(* CoDeSys 2.3 export: A_CONV.EXP *)

(* POU A_CONVER, CFC *)
FUNCTION_BLOCK A_CONVER
VAR_INPUT
	IN : REAL;
	IN_MIN : REAL := 4;
	IN_MAX : REAL := 20;
	OUT_MIN : REAL := 4;
	OUT_MAX : REAL := 20;
END_VAR
VAR_OUTPUT
	OUT : WORD;

END_VAR
VAR
	LIN1: LIN_TRAFO;
END_VAR
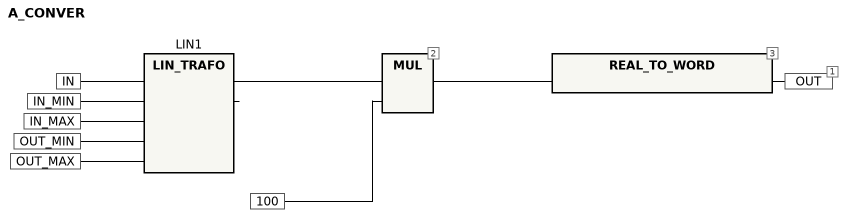
_CFC_ (* Continuous Function Chart, elements in execution order *)
#0 LIN1:LIN_TRAFO(IN, IN_MIN, IN_MAX, OUT_MIN, OUT_MAX)
#1 OUT <= #3
#2 MUL(#0.out 1, 100)
#3 REAL_TO_WORD(#2)
_END_CFC_
END_FUNCTION_BLOCK
